(* CODESYS project ESA_ZadataQ2_2015-16.project
   CustomField04_name: CustomField04
   CustomField06_name: CustomField06
   CustomField07_name: CustomField07
   CustomField09_name: CustomField09
   CustomField08_name: CustomField08
   CustomField02_name: CustomField02
   CustomField10_name: CustomField10
   CustomField01_name: CustomField01
   CustomField03_name: CustomField03
   CustomField05_name: CustomField05

Project tree, tasks and I/O mapping:
  MyController : TM238LFDC24DT, Schneider Electric, order no. TM238LFDC24DT, version 2.0.31.8
    application Application
      task MAST (cyclic, interval 20 ms, priority 15, watchdog 100 ms x 1) calls POU
      global variables GVL
      program POU [LD]
      function HiddenPOU [ST]
    Embedded Functions
      IO : IO, Schneider Electric, version 2.0.31.8
          input  Application.POU.Tipkalo3 : BOOL  // IW0.I8
          input  Application.POU.Tipkalo2 : BOOL  // IW0.I9
          input  Application.POU.Tipkalo1 : BOOL  // IW0.I10
          input  Application.POU.Sklopka1 : BOOL  // IW0.I11
          input  Application.POU.Sklopka2 : BOOL  // IW0.I12
          output Application.POU.Zelena1 : BOOL  // QW0.Q4
          output Application.POU.Zuta1 : BOOL  // QW0.Q5
          output Application.POU.Crvena1 : BOOL  // QW0.Q6
          output Application.POU.Zelena2 : BOOL  // QW0.Q7
          output Application.POU.Zuta2 : BOOL  // QW0.Q8
          output Application.POU.Crvena2 : BOOL  // QW0.Q9
          unmapped channels: IW0, QW0
      HSC : HSC, Schneider Electric, version 2.0.31.8
        HSC
      PTO_PWM : PTO_PWM, Schneider Electric, version 2.0.31.8
        PTO_PWM
    Serial Line 2
      SoMachine_Network_Manager : SoMachine-Network_Manager, Schneider Electric, version 2.0.1.10
    CAN
    Serial Line 1
      Modbus_Manager : Modbus_Manager, Schneider Electric, version 2.0.1.12
  MachineLayoutPicture
*)

// MyController/Application/GVL
VAR_GLOBAL
END_VAR

// MyController/Application/POU
PROGRAM POU
VAR_INPUT
	Sklopka1 :BOOL;
	Sklopka2 :BOOL;
	Tipkalo1 :BOOL;
	Tipkalo2 :BOOL;
	Tipkalo3 :BOOL;
	brojka :INT;
END_VAR
VAR_OUTPUT
	Zelena1 :BOOL;
	Zelena2 :BOOL;
	Crvena1 :BOOL;
	Crvena2 :BOOL;
	Zuta1 :BOOL;
	Zuta2 :BOOL;
	
END_VAR

VAR
		
	C1 : CTUD;      					//counter 1
	Blink_Gen : BLINK ;					//blinkani signal
	Time_blink: TIME := T#0.01S;			//vrijeme blinkanja
	Time_untillTipkalo: TIME;  			//vrijeme od zadnjeg pritiska tipkala
	trenutnibroj: WORD;					//trenutni broj na brojilu
	kriticnibroj:WORD := 5; 			//broj nakon kojeg idu promjene (5) 
	Brojilo: TON;						//tajmer	
	pocetiBlinkanje: BOOL; 				//bool koji govori da je isteklo vrijeme i da treba poceti blinkati!!!!
	blink_signal: BOOL;					//blinkani signal (ukljucuje se nakon sto je isteklo poitrebno vrijeme, inace je 0
END_VAR

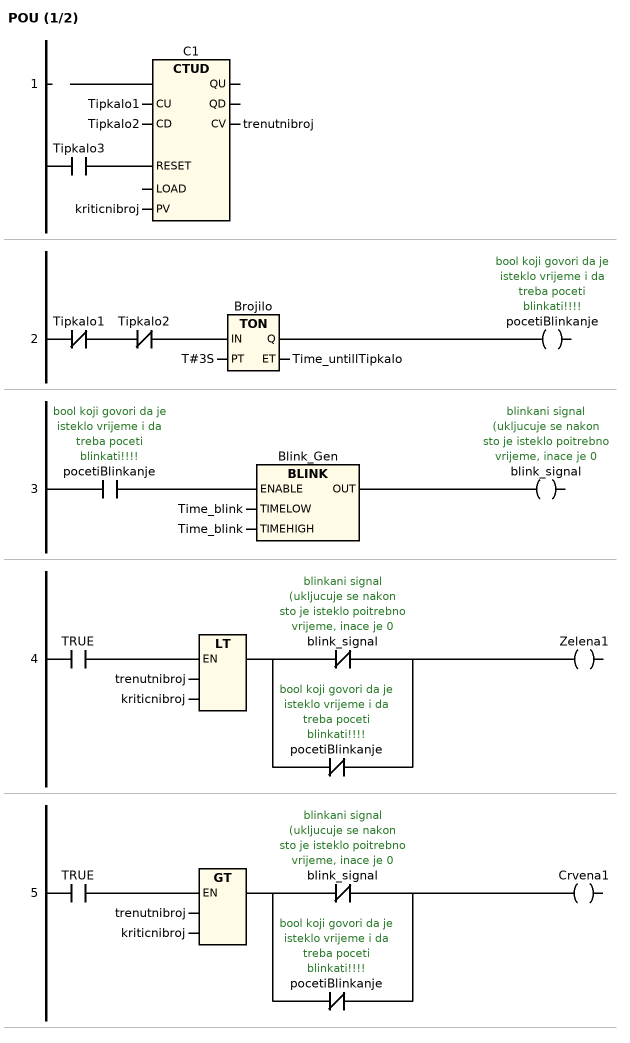
// NETWORK 1
//   C1: counter 1
//   kriticnibroj: broj nakon kojeg idu promjene (5)
//   trenutnibroj: trenutni broj na brojilu
C1(CU := Tipkalo1, CD := Tipkalo2, RESET := Tipkalo3, PV := kriticnibroj, CV => trenutnibroj); // CTUD

// NETWORK 2
//   Brojilo: tajmer
//   Time_untillTipkalo: vrijeme od zadnjeg pritiska tipkala
//   pocetiBlinkanje: bool koji govori da je isteklo vrijeme i da treba poceti blinkati!!!!
Brojilo(IN := NOT Tipkalo1 AND NOT Tipkalo2, PT := T#3S, ET => Time_untillTipkalo); // TON
pocetiBlinkanje := Brojilo.Q;

// NETWORK 3
//   Blink_Gen: blinkani signal
//   pocetiBlinkanje: bool koji govori da je isteklo vrijeme i da treba poceti blinkati!!!!
//   Time_blink: vrijeme blinkanja
//   blink_signal: blinkani signal (ukljucuje se nakon sto je isteklo poitrebno vrijeme, inace je 0
Blink_Gen(ENABLE := pocetiBlinkanje, TIMELOW := Time_blink, TIMEHIGH := Time_blink); // BLINK
blink_signal := Blink_Gen.OUT;

// NETWORK 4
//   trenutnibroj: trenutni broj na brojilu
//   kriticnibroj: broj nakon kojeg idu promjene (5)
//   blink_signal: blinkani signal (ukljucuje se nakon sto je isteklo poitrebno vrijeme, inace je 0
//   pocetiBlinkanje: bool koji govori da je isteklo vrijeme i da treba poceti blinkati!!!!
Zelena1 := trenutnibroj < kriticnibroj AND (NOT blink_signal OR NOT pocetiBlinkanje);

// NETWORK 5
//   trenutnibroj: trenutni broj na brojilu
//   kriticnibroj: broj nakon kojeg idu promjene (5)
//   blink_signal: blinkani signal (ukljucuje se nakon sto je isteklo poitrebno vrijeme, inace je 0
//   pocetiBlinkanje: bool koji govori da je isteklo vrijeme i da treba poceti blinkati!!!!
Crvena1 := trenutnibroj > kriticnibroj AND (NOT blink_signal OR NOT pocetiBlinkanje);

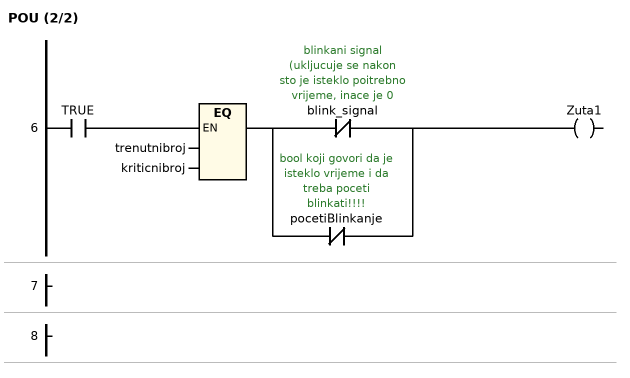
// NETWORK 6
//   trenutnibroj: trenutni broj na brojilu
//   kriticnibroj: broj nakon kojeg idu promjene (5)
//   blink_signal: blinkani signal (ukljucuje se nakon sto je isteklo poitrebno vrijeme, inace je 0
//   pocetiBlinkanje: bool koji govori da je isteklo vrijeme i da treba poceti blinkati!!!!
Zuta1 := trenutnibroj = kriticnibroj AND (NOT blink_signal OR NOT pocetiBlinkanje);

// NETWORK 7

// NETWORK 8

END_PROGRAM

// MyController/Application/HiddenPOU
FUNCTION HiddenPOU : BOOL

VAR_INPUT
	pHiddenFunc: POINTER TO WORD;
END_VAR
VAR
	pRead: POINTER TO BYTE;
	pWrite: POINTER TO BYTE;
END_VAR

pRead := pHiddenFunc + 400;
pWrite := pHiddenFunc + 4400;
HiddenPOU := TRUE;

END_FUNCTION
